// TIA Portal V19 export
DATA_BLOCK "REGENRATION DB"   // DB79
{ S7_Optimized_Access := 'TRUE' }
// stored: MemoryReserve 100
   VAR
      "REGRNRATION START" : Bool;
      "REGRNRATION BUFF" : Int;
   END_VAR
   VAR RETAIN
      "SET VALVE" : Struct
         "SOFTENER BACKWASH" : Int;
         "SALT SUCTION" : Int;
         "SALT HOLDING" : Int;
         "SLOW RINSE WASH" : Int;
         "FAST RINS WASH" : Int;
      END_STRUCT;
   END_VAR
   VAR
      "PV VALVE" : Struct
         "SOFTENER BACKWASH" : Int;
         "SALT SUCTION" : Int;
         "SALT HOLDING" : Int;
         "SLOW RINSE WASH" : Int;
         "FAST RINS WASH" : Int;
      END_STRUCT;
   END_VAR
BEGIN
END_DATA_BLOCK
